TYPE VelocityCtrl_typ :
	STRUCT
		Input	: VelocityCtrl_Input_typ ;
		Output	: VelocityCtrl_Output_typ ;
	END_STRUCT
END_TYPE

(* stored: Version 1.1.0.1, ProductVersion 3.1.4024.3
   DUT VelocityCtrl_typ: Id {9aa8f6b1-6f4a-432c-9b9b-263ab70a0b14} *)
